{attribute 'qualified_only'}
{attribute 'strict'}
TYPE E_Z4_Step :
(
	(* special steps *)
	NoStep := -32767,		// nessuno step
	Unknown := -32000,		// step sconosciuto
	
	(* Error steps *)
	NeOrError := -990,		// non abilitata o in errore
	Recovering := -980,		// azzeramento errori
		
	(* Stop *)
	Stop := 0,				// S0, stop
	
	(* Cycle *)
	Ready := 100,			// S1, pronto a ricevere pezzo
	MoveToDrill := 120,		// S2, avanza il nastro fino al trapano
	Drilling := 140,		// S3, lavorazione con il trapano
	WaitZ5Ready := 160,		// S4, attende che Z5 sia ready
	MoveToZ5 := 180,		// S5, avanza il nastro fino a Z5

	Done := 800,			// Ciclo concluso
	
	(* Stopping *)
	Stopping := 900	
);
END_TYPE
//  NoStep = '-32767'
//  Unknown = '-32000'
//  NeOrError = '-990'
//  Recovering = '-980'

(* stored: Version 1.1.0.1
   EnumerationTextList E_Z4_Step: Id {6f8e1620-d172-04b8-0ce6-bbba1b30220e} *)
